(* IEC 61131-3 sources: ATCMcontrol_Engineering/src/Target/ATHW119/Libs/ATCM_IEC1131_3/table_26, 4 files *)

(* ---- and.st ---- *)
(*[[
    UserURL= "ATCMfile:AND.htm"
]]*)

FUNCTION AND : ANY_BIT
VAR_INPUT
    IN1 : ANY_BIT;
END_VAR
VAR_IN_EXT
    IN2 : ANY_BIT;
END_VAR

inline AND

END_FUNCTION

(* ---- not.st ---- *)
(*[[
    UserURL= "ATCMfile:NOT.htm"
]]*)

FUNCTION NOT : ANY_BIT
VAR_INPUT
    IN : ANY_BIT;
END_VAR

inline NOT

END_FUNCTION

(* ---- or.st ---- *)
(*[[
    UserURL= "ATCMfile:OR.htm"
]]*)

FUNCTION OR : ANY_BIT
VAR_INPUT
    IN1 : ANY_BIT;
END_VAR
VAR_IN_EXT
    IN2 : ANY_BIT;
END_VAR

inline OR

END_FUNCTION

(* ---- xor.st ---- *)
(*[[
    UserURL= "ATCMfile:XOR.htm"
]]*)

FUNCTION XOR : ANY_BIT
VAR_INPUT
    IN1 : ANY_BIT;
END_VAR
VAR_IN_EXT
    IN2 : ANY_BIT;
END_VAR

inline XOR

END_FUNCTION
